RoboDK station: Shape_detection.rdk

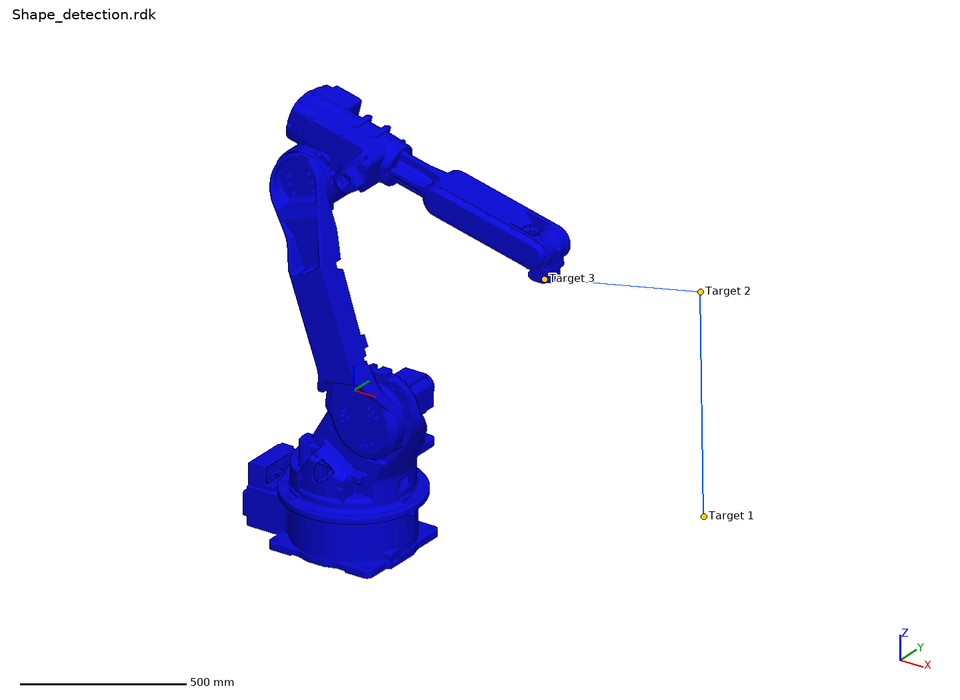
[picture v0: the station drawn from its stored meshes, robots at their saved joint values, targets as dots, program paths as lines]
Station Shape_detection (saved by RoboDK 5.6.3). Poses are relative to the parent item; angles as X-Y-Z fixed-axis rotations.
  - frame Motoman HP20D Base at (0, 0, 505) mm
    - robot Motoman HP20D: 6 axes, payload 20 kg, reach 1717 mm, repeatability 0.06 mm, weight 268 kg
        modified DH rows (alpha deg, a mm, theta deg, d mm): 0, 0, 0, 505; -90, 150, -90, 0; 0, 760, 0, 0; -90, 140, 0, 795; 90, 0, 90, 0; -90, 0, 0, 105
        base shift (0, 0, -505) mm
        joint limits [-180, -110, -165, -200, -50, -360] to [180, 155, 255, 200, 230, 360]; home [0, 0, 0, 0, 0, 0]; saved at [0, -19.463, -32.509, 0, 13.046, 0]
    - target Target 3 (Cartesian target) at (702.85, 0, 568.5) mm, rotated rx -180 ry 0 rz 0 deg; joints [0, -19.463, -32.509, 0, 13.046, 0] of Motoman HP20D
    - target Target 2 (Cartesian target) at (1274.1, 0, 685.56) mm, rotated rx -180 ry 0 rz 0 deg; joints [0, 25.188, 22.518, 0, 2.67, 0] of Motoman HP20D
    - target Target 1 (Cartesian target) at (1286.04, 0, -61.38) mm, rotated rx -180 ry 0 rz 0 deg; joints [0, 42.639, -7.032, 0, 49.671, 0] of Motoman HP20D
  - program Prog1 (4 instructions, listed below)
  - Python program Prog2 (listed below)
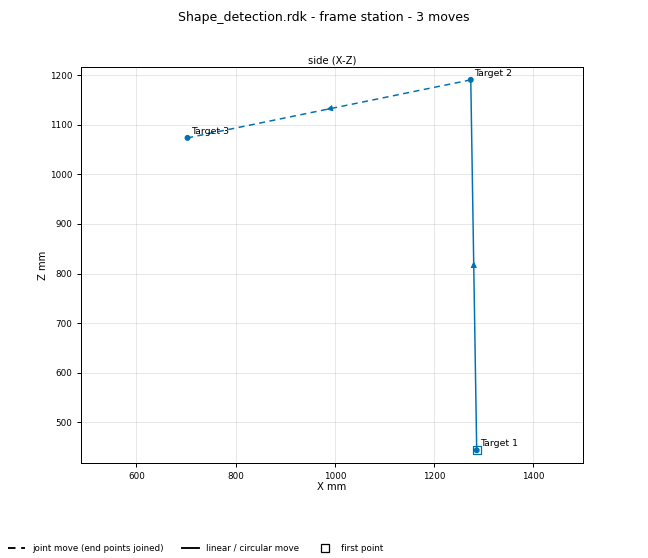
[picture p0: tool path of Shape_detection.rdk in frame station, 3 of 3 moves have a stored position in this frame; points joined in program order, loops and branches not executed]

--- program Prog1 (robot Motoman HP20D) ---
  Est. Ref.: Motoman HP20D Base
  MoveL (Target 1)
  MoveL (Target 2)
  MoveJ (Target 3)

--- Python program Prog2 ---
from robolink import *    # RoboDK's API
from robodk import *      # Math toolbox for robots

RDK = Robolink()
robot = RDK.Item('', ITEM_TYPE_ROBOT)

#Comprobación de movimientos
target = RDK.Item('Target 1')
target2 = RDK.Item('Target 2')
target3 = RDK.Item('Target 3')
program = RDK.Item('Prog1')
target_pose = target.Pose()
xyz_ref = target_pose.Pos()

import cv2 as cv
import numpy as np
import imutils

def real_time_shape(show):
    cap_video = cv.VideoCapture(0)

    while True:
        _, frame = cap_video.read()
        frameG = cv.cvtColor(frame, cv.COLOR_BGR2GRAY)
        edges = cv.Canny(frameG, 200, 200)
        thresh = cv.threshold(frameG, 127, 255, cv.THRESH_BINARY)[1]
        shapes = shapeDetector(thresh, frame.copy())

        if show:
            cv.imshow('Original Image', frame)
            cv.imshow('Edges', edges)
            cv.imshow('Threshold', thresh)
            cv.imshow('Shapes', shapes)

        key = cv.waitKey(1)
        if key == 27:
            break

    cap_video.release()
    cv.destroyAllWindows()

def shapeDetector(image, origimage):
    resized = imutils.resize(image, width=300)
    ratio = image.shape[0] / float(resized.shape[0])
    contours = cv.findContours(resized.copy(), cv.RETR_EXTERNAL, cv.CHAIN_APPROX_SIMPLE)[0]

    for cntour in contours:
        shape = detect(cntour)
        M = cv.moments(cntour)
        if M["m00"] == 0:
            cX, cY = 0, 0
        else:
            cX = int((M["m10"] / M["m00"]) * ratio)
            cY = int((M["m01"] / M["m00"]) * ratio)
        cntour = cntour.astype("float") * ratio
        cntour = cntour.astype("int")
        cv.drawContours(origimage, [cntour], -1, (34, 0, 156), 2)
        cv.putText(origimage, shape, (cX, cY), cv.FONT_HERSHEY_SIMPLEX,
                   0.5, (255, 255, 255), 2)
    return origimage

def detect(c):
    shape = "unidentified"
    peri = cv.arcLength(c, True)
    approx = cv.approxPolyDP(c, 0.04 * peri, True)
    if len(approx) == 3:
        shape = "triangle"
        robot.MoveJ(target)
        robot.RunInstruction('Program_Done')
    elif len(approx) == 4:
        (_, _, w, h) = cv.boundingRect(approx)
        ar = w / float(h)
        if 0.95 <= ar <= 1.05:  # Si es cuadrado
            shape = "square"
            robot.MoveJ(target2)
            robot.RunInstruction('Program_Done')
        else:  # Si es rectángulo
            shape = "rectangle"
            robot.MoveJ(target3)
            robot.RunInstruction('Program_Done')
    else:
        shape = "circle"
        program.RunProgram()
        robot.RunInstruction('Program_Done')
    return shape

if __name__ == "__main__":
    real_time_shape(1)
